// TIA Portal V21 export
VAR_GLOBAL   // PLC tag table "Default tag table"
   Start AT %M0.0 : Bool;
   Motor AT %Q0.1 : Bool;
   Stop AT %M0.1 : Bool;
   Foward AT %M0.2 : Bool;
   Revense AT %M0.3 : Bool;
   RunFoward AT %Q0.2 : Bool;
   RunRevense AT %Q0.3 : Bool;
   Lamp AT %Q0.4 : Bool;
   Ready AT %M1.0 : Bool;
   Alarm AT %M1.1 : Bool;
END_VAR
